{attribute 'qualified_only'}
{attribute 'strict'}
TYPE E_Xelectrix_BatteryState :
(
	eNoDataReceived := 0,
	eOff := 1,
	eStartUp := 2,
	eBalancing := 3,
	eReady := 4,
	eOperating := 5,
	eError := 6
);
END_TYPE

(* stored: Version 1.1.0.1, ProductVersion 3.1.4024.9
   DUT E_Xelectrix_BatteryState: Id {f64a8189-0a7f-4eb0-acae-cded31d068fc} *)
